FUNCTION TryConvert_UINT_TO_BYTE : BOOL
VAR_INPUT
	in : UINT;
	out : REFERENCE TO BYTE;
END_VAR

IF in > DatatypeLimits.MAX_VALUE_OF_UINT_WHICH_CAN_BE_HELD_IN_A_BYTE THEN
	RETURN;
END_IF

out := UINT_TO_BYTE(in);
TryConvert_UINT_TO_BYTE := TRUE;

END_FUNCTION

(* stored: Version 1.1.0.1, ProductVersion 3.1.4024.12
   POU TryConvert_UINT_TO_BYTE: Id {60a77519-5c86-4bed-b3c1-05bbb1612155}, SpecialFunc None *)
